FUNCTION_BLOCK VVL_HMI (* HMI and Local Multicast elements for testing a Valve view. *)
  (* Standard: IEC 61499; Classification: HMI; ApplicationDomain: Process Control; Function: Test; Type: ON/OFF Valve *)
  (* Version 0.0, 2006-07-28, JHC, Holobloc Inc *)
  (* Compiler header: package fb.rt.batch; import fb.rt.net.*; import fb.rt.gui.*; import fb.rt.hmi.*; import fb.rt.mva.FBMVCD; *)
  (* Compiler classdef: public class VVL_HMI extends FBMVCD *)
  (* Compiler Java Sun JDK 1.5.0 *)
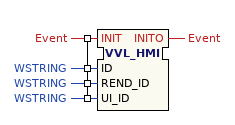
  EVENT_INPUT
    INIT WITH REND_ID, UI_ID, ID; (* Initialization Request *)
  END_EVENT
  EVENT_OUTPUT
    INITO; (* Initialization Confirm *)
  END_EVENT
  VAR_INPUT
    ID : WSTRING; (* Label for HMI elements, default = FB instance name *)
    REND_ID : WSTRING; (* Local Channel ID for rendering data *)
    UI_ID : WSTRING; (* Local Channel ID for valve state publication *)
  END_VAR
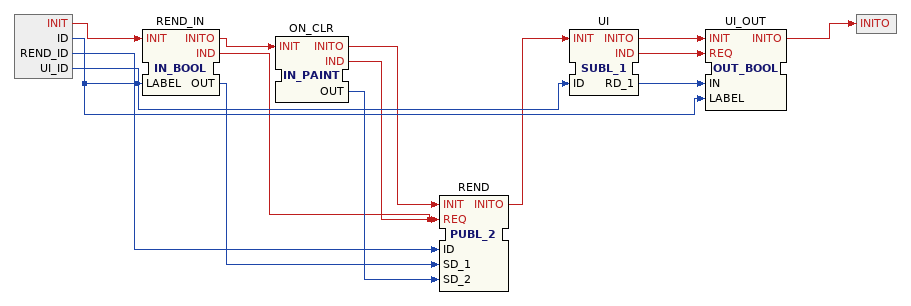
  FBS
    UI : SUBL_1;
    REND : PUBL_2;
    REND_IN : IN_BOOL;
    UI_OUT : OUT_BOOL;
    ON_CLR : IN_PAINT; (* Valve ON Paint pattern key *)
  END_FBS
  EVENT_CONNECTIONS
    INIT TO REND_IN.INIT;
    REND.INITO TO UI.INIT;
    UI.INITO TO UI_OUT.INIT;
    UI.IND TO UI_OUT.REQ;
    UI_OUT.INITO TO INITO;
    REND_IN.INITO TO ON_CLR.INIT;
    ON_CLR.INITO TO REND.INIT;
    ON_CLR.IND TO REND.REQ;
    REND_IN.IND TO REND.REQ;
  END_CONNECTIONS
  DATA_CONNECTIONS
    REND_ID TO REND.ID;
    UI_ID TO UI.ID;
    ID TO REND_IN.LABEL;
    REND_IN.OUT TO REND.SD_1;
    UI.RD_1 TO UI_OUT.IN;
    ID TO UI_OUT.LABEL;
    ON_CLR.OUT TO REND.SD_2;
  END_CONNECTIONS
END_FUNCTION_BLOCK
